   1:  PR[GP1:91,2] = PR[GP1:90,2] + -27.473;
   1:L PR[91] R[100]mm/sec CNT100;
   1:  PR[GP1:91,1] = PR[GP1:90,1] + 0.138;
   1:  PR[GP1:91,2] = PR[GP1:90,2] + -27.866;
   1:L PR[91] R[100]mm/sec CNT100;
   1:  PR[GP1:91,1] = PR[GP1:90,1] + 2.042;
   1:  PR[GP1:91,2] = PR[GP1:90,2] + -27.743;
   1:L PR[91] R[100]mm/sec CNT100;
   1:  PR[GP1:91,1] = PR[GP1:90,1] + 3.999;
   1:  PR[GP1:91,2] = PR[GP1:90,2] + -27.362;
   1:L PR[91] R[100]mm/sec CNT100;
   1:  PR[GP1:91,1] = PR[GP1:90,1] + 7.084;
   1:  PR[GP1:91,2] = PR[GP1:90,2] + -26.955;
   1:L PR[91] R[100]mm/sec CNT100;
   1:  PR[GP1:91,1] = PR[GP1:90,1] + 10.547;
   1:  PR[GP1:91,2] = PR[GP1:90,2] + -25.597;
   1:L PR[91] R[100]mm/sec CNT100;
   1:  PR[GP1:91,1] = PR[GP1:90,1] + 13.465;
   1:  PR[GP1:91,2] = PR[GP1:90,2] + -24.388;
   1:L PR[91] R[100]mm/sec CNT100;
   1:  PR[GP1:91,1] = PR[GP1:90,1] + 16.487;
   1:  PR[GP1:91,2] = PR[GP1:90,2] + -22.246;
   1:L PR[91] R[100]mm/sec CNT100;
   1:  PR[GP1:91,1] = PR[GP1:90,1] + 19.071;
   1:  PR[GP1:91,2] = PR[GP1:90,2] + -20.263;
   1:L PR[91] R[100]mm/sec CNT100;
   1:  PR[GP1:91,1] = PR[GP1:90,1] + 21.139;
   1:  PR[GP1:91,2] = PR[GP1:90,2] + -17.946;
   1:L PR[91] R[100]mm/sec CNT100;
   1:  PR[GP1:91,1] = PR[GP1:90,1] + 23.096;
   1:  PR[GP1:91,2] = PR[GP1:90,2] + -15.395;
   1:L PR[91] R[100]mm/sec CNT100;
   1:  PR[GP1:91,1] = PR[GP1:90,1] + 24.605;
   1:  PR[GP1:91,2] = PR[GP1:90,2] + -12.804;
   1:L PR[91] R[100]mm/sec CNT100;
   1:  PR[GP1:91,1] = PR[GP1:90,1] + 25.817;
   1:  PR[GP1:91,2] = PR[GP1:90,2] + -9.880;
   1:L PR[91] R[100]mm/sec CNT100;
   1:  PR[GP1:91,1] = PR[GP1:90,1] + 26.838;
   1:  PR[GP1:91,2] = PR[GP1:90,2] + -6.844;
   1:L PR[91] R[100]mm/sec CNT100;
   1:  PR[GP1:91,1] = PR[GP1:90,1] + 27.222;
   1:  PR[GP1:91,2] = PR[GP1:90,2] + -3.380;
   1:L PR[91] R[100]mm/sec CNT100;
   1:  PR[GP1:91,1] = PR[GP1:90,1] + 27.629;
   1:  PR[GP1:91,2] = PR[GP1:90,2] + -0.292;
   1:L PR[91] R[100]mm/sec CNT100;
   1:  PR[GP1:91,1] = PR[GP1:90,1] + 27.296;
   1:  PR[GP1:91,2] = PR[GP1:90,2] + 2.903;
   1:L PR[91] R[100]mm/sec CNT100;
   1:  PR[GP1:91,1] = PR[GP1:90,1] + 26.887;
   1:  PR[GP1:91,2] = PR[GP1:90,2] + 6.009;
   1:L PR[91] R[100]mm/sec CNT100;
   1:  PR[GP1:91,1] = PR[GP1:90,1] + 25.954;
   1:  PR[GP1:91,2] = PR[GP1:90,2] + 8.948;
   1:L PR[91] R[100]mm/sec CNT100;
   1:  PR[GP1:91,1] = PR[GP1:90,1] + 24.744;
   1:  PR[GP1:91,2] = PR[GP1:90,2] + 11.869;
   1:L PR[91] R[100]mm/sec CNT100;
   1:  PR[GP1:91,1] = PR[GP1:90,1] + 23.230;
   1:  PR[GP1:91,2] = PR[GP1:90,2] + 14.583;
   1:L PR[91] R[100]mm/sec CNT100;
   1:  PR[GP1:91,1] = PR[GP1:90,1] + 21.280;
   1:  PR[GP1:91,2] = PR[GP1:90,2] + 17.124;
   1:L PR[91] R[100]mm/sec CNT100;
   1:  PR[GP1:91,1] = PR[GP1:90,1] + 19.067;
   1:  PR[GP1:91,2] = PR[GP1:90,2] + 19.643;
   1:L PR[91] R[100]mm/sec CNT100;
   1:  PR[GP1:91,1] = PR[GP1:90,1] + 16.487;
   1:  PR[GP1:91,2] = PR[GP1:90,2] + 21.622;
   1:L PR[91] R[100]mm/sec CNT100;
   1:  PR[GP1:91,1] = PR[GP1:90,1] + 13.451;
   1:  PR[GP1:91,2] = PR[GP1:90,2] + 23.772;
   1:L PR[91] R[100]mm/sec CNT100;
   1:  PR[GP1:91,1] = PR[GP1:90,1] + 10.457;
   1:  PR[GP1:91,2] = PR[GP1:90,2] + 25.012;
   1:L PR[91] R[100]mm/sec CNT100;
   1:  PR[GP1:91,1] = PR[GP1:90,1] + 6.989;
   1:  PR[GP1:91,2] = PR[GP1:90,2] + 26.356;
   1:L PR[91] R[100]mm/sec CNT100;
   1:  PR[GP1:91,1] = PR[GP1:90,1] + 3.774;
   1:  PR[GP1:91,2] = PR[GP1:90,2] + 26.779;
   1:L PR[91] R[100]mm/sec CNT100;
   1:  PR[GP1:91,1] = PR[GP1:90,1] + 0.078;
   1:  PR[GP1:91,2] = PR[GP1:90,2] + 27.237;
   1:L PR[91] R[100]mm/sec CNT100;
   1:  PR[91] = PR[90];
   1:  PR[GP1:91,1] = PR[GP1:90,1] + -2.874;
   1:  PR[GP1:91,2] = PR[GP1:90,2] + 26.871;
   1:  PR[GP1:91,3] = PR[GP1:90,3] + 77.775;
   1:L PR[91] R[100]mm/sec CNT100;
   1:  PR[GP1:91,1] = PR[GP1:90,1] + -6.879;
   1:  PR[GP1:91,2] = PR[GP1:90,2] + 26.344;
   1:L PR[91] R[100]mm/sec CNT100;
   1:  PR[GP1:91,1] = PR[GP1:90,1] + -9.647;
   1:  PR[GP1:91,2] = PR[GP1:90,2] + 25.271;
   1:L PR[91] R[100]mm/sec CNT100;
   1:  PR[GP1:91,1] = PR[GP1:90,1] + -13.376;
   1:  PR[GP1:91,2] = PR[GP1:90,2] + 23.726;
   1:L PR[91] R[100]mm/sec CNT100;
   1:  PR[GP1:91,1] = PR[GP1:90,1] + -15.799;
   1:  PR[GP1:91,2] = PR[GP1:90,2] + 22.010;
   1:L PR[91] R[100]mm/sec CNT100;
   1:  PR[GP1:91,1] = PR[GP1:90,1] + -19.016;
   1:  PR[GP1:91,2] = PR[GP1:90,2] + 19.543;
   1:L PR[91] R[100]mm/sec CNT100;
   1:  PR[GP1:91,1] = PR[GP1:90,1] + -20.663;
   1:  PR[GP1:91,2] = PR[GP1:90,2] + 17.697;
   1:L PR[91] R[100]mm/sec CNT100;
   1:  PR[GP1:91,1] = PR[GP1:90,1] + -23.111;
   1:  PR[GP1:91,2] = PR[GP1:90,2] + 14.505;
   1:L PR[91] R[100]mm/sec CNT100;
   1:  PR[GP1:91,1] = PR[GP1:90,1] + -24.313;
   1:  PR[GP1:91,2] = PR[GP1:90,2] + 12.443;
   1:L PR[91] R[100]mm/sec CNT100;
   1:  PR[GP1:91,1] = PR[GP1:90,1] + -25.837;
   1:  PR[GP1:91,2] = PR[GP1:90,2] + 8.764;
   1:L PR[91] R[100]mm/sec CNT100;
   1:  PR[GP1:91,1] = PR[GP1:90,1] + -26.650;
   1:  PR[GP1:91,2] = PR[GP1:90,2] + 6.347;
   1:L PR[91] R[100]mm/sec CNT100;
   1:  PR[GP1:91,1] = PR[GP1:90,1] + -26.957;
   1:  PR[GP1:91,2] = PR[GP1:90,2] + 3.574;
   1:L PR[91] R[100]mm/sec CNT100;
   1:  PR[GP1:91,1] = PR[GP1:90,1] + -27.472;
   1:  PR[GP1:91,2] = PR[GP1:90,2] + -0.332;
   1:L PR[91] R[100]mm/sec CNT100;
   1:  PR[GP1:91,1] = PR[GP1:90,1] + -27.207;
   1:  PR[GP1:91,2] = PR[GP1:90,2] + -2.875;
   1:L PR[91] R[100]mm/sec CNT100;
   1:  PR[GP1:91,1] = PR[GP1:90,1] + -26.691;
   1:  PR[GP1:91,2] = PR[GP1:90,2] + -6.797;
   1:L PR[91] R[100]mm/sec CNT100;
   1:  PR[GP1:91,1] = PR[GP1:90,1] + -25.949;
   1:  PR[GP1:91,2] = PR[GP1:90,2] + -9.137;
   1:L PR[91] R[100]mm/sec CNT100;
   1:  PR[GP1:91,1] = PR[GP1:90,1] + -24.426;
   1:  PR[GP1:91,2] = PR[GP1:90,2] + -12.814;
   1:L PR[91] R[100]mm/sec CNT100;
   1:  PR[GP1:91,1] = PR[GP1:90,1] + -23.218;
   1:  PR[GP1:91,2] = PR[GP1:90,2] + -14.979;
   1:L PR[91] R[100]mm/sec CNT100;
   1:  PR[GP1:91,1] = PR[GP1:90,1] + -20.776;
   1:  PR[GP1:91,2] = PR[GP1:90,2] + -18.162;
   1:L PR[91] R[100]mm/sec CNT100;
   1:  PR[GP1:91,1] = PR[GP1:90,1] + -19.001;
   1:  PR[GP1:91,2] = PR[GP1:90,2] + -20.182;
   1:L PR[91] R[100]mm/sec CNT100;
   1:  PR[GP1:91,1] = PR[GP1:90,1] + -17.808;
   1:  PR[GP1:91,2] = PR[GP1:90,2] + -21.138;
   1:L PR[91] R[100]mm/sec CNT100;
   1:  PR[GP1:91,1] = PR[GP1:90,1] + -14.562;
   1:  PR[GP1:91,2] = PR[GP1:90,2] + -23.628;
   1:L PR[91] R[100]mm/sec CNT100;
   1:  PR[GP1:91,1] = PR[GP1:90,1] + -13.334;
   1:  PR[GP1:91,2] = PR[GP1:90,2] + -24.378;
   1:L PR[91] R[100]mm/sec CNT100;
   1:  PR[GP1:91,1] = PR[GP1:90,1] + -9.628;
   1:  PR[GP1:91,2] = PR[GP1:90,2] + -25.913;
   1:L PR[91] R[100]mm/sec CNT100;
   1:  PR[GP1:91,1] = PR[GP1:90,1] + -6.838;
   1:  PR[GP1:91,2] = PR[GP1:90,2] + -26.978;
   1:L PR[91] R[100]mm/sec CNT100;
   1:  PR[GP1:91,1] = PR[GP1:90,1] + -3.689;
   1:  PR[GP1:91,2] = PR[GP1:90,2] + -27.362;
   1:L PR[91] R[100]mm/sec CNT100;
   1:  PR[GP1:91,1] = PR[GP1:90,1] + 0.136;
   1:  PR[GP1:91,2] = PR[GP1:90,2] + -27.866;
   1:L PR[91] R[100]mm/sec CNT100;
   1:  PR[GP1:91,1] = PR[GP1:90,1] + 1.630;
   1:  PR[GP1:91,2] = PR[GP1:90,2] + -27.769;
   1:L PR[91] R[100]mm/sec CNT100;
   1:  PR[GP1:91,1] = PR[GP1:90,1] + 3.202;
   1:  PR[GP1:91,2] = PR[GP1:90,2] + -27.463;
   1:L PR[91] R[100]mm/sec CNT100;
   1:  PR[GP1:91,1] = PR[GP1:90,1] + 7.110;
   1:  PR[GP1:91,2] = PR[GP1:90,2] + -26.948;
   1:L PR[91] R[100]mm/sec CNT100;
   1:  PR[GP1:91,1] = PR[GP1:90,1] + 9.876;
   1:  PR[GP1:91,2] = PR[GP1:90,2] + -25.864;
   1:L PR[91] R[100]mm/sec CNT100;
   1:  PR[GP1:91,1] = PR[GP1:90,1] + 13.544;
   1:  PR[GP1:91,2] = PR[GP1:90,2] + -24.344;
   1:L PR[91] R[100]mm/sec CNT100;
   1:  PR[GP1:91,1] = PR[GP1:90,1] + 15.956;
   1:  PR[GP1:91,2] = PR[GP1:90,2] + -22.634;
   1:L PR[91] R[100]mm/sec CNT100;
   1:  PR[GP1:91,1] = PR[GP1:90,1] + 19.173;
   1:  PR[GP1:91,2] = PR[GP1:90,2] + -20.167;
   1:L PR[91] R[100]mm/sec CNT100;
   1:  PR[GP1:91,1] = PR[GP1:90,1] + 20.820;
   1:  PR[GP1:91,2] = PR[GP1:90,2] + -18.321;
   1:L PR[91] R[100]mm/sec CNT100;
   1:  PR[GP1:91,1] = PR[GP1:90,1] + 23.269;
   1:  PR[GP1:91,2] = PR[GP1:90,2] + -15.129;
   1:L PR[91] R[100]mm/sec CNT100;
   1:  PR[GP1:91,1] = PR[GP1:90,1] + 24.470;
   1:  PR[GP1:91,2] = PR[GP1:90,2] + -13.066;
   1:L PR[91] R[100]mm/sec CNT100;
   1:  PR[GP1:91,1] = PR[GP1:90,1] + 25.994;
   1:  PR[GP1:91,2] = PR[GP1:90,2] + -9.387;
   1:L PR[91] R[100]mm/sec CNT100;
   1:  PR[GP1:91,1] = PR[GP1:90,1] + 26.807;
   1:  PR[GP1:91,2] = PR[GP1:90,2] + -6.971;
   1:L PR[91] R[100]mm/sec CNT100;
   1:  PR[GP1:91,1] = PR[GP1:90,1] + 27.114;
   1:  PR[GP1:91,2] = PR[GP1:90,2] + -4.198;
   1:L PR[91] R[100]mm/sec CNT100;
   1:  PR[GP1:91,1] = PR[GP1:90,1] + 27.629;
   1:  PR[GP1:91,2] = PR[GP1:90,2] + -0.292;
   1:L PR[91] R[100]mm/sec CNT100;
   1:  PR[GP1:91,1] = PR[GP1:90,1] + 27.364;
   1:  PR[GP1:91,2] = PR[GP1:90,2] + 2.254;
   1:L PR[91] R[100]mm/sec CNT100;
   1:  PR[GP1:91,1] = PR[GP1:90,1] + 26.847;
   1:  PR[GP1:91,2] = PR[GP1:90,2] + 6.176;
   1:L PR[91] R[100]mm/sec CNT100;
   1:  PR[GP1:91,1] = PR[GP1:90,1] + 26.104;
   1:  PR[GP1:91,2] = PR[GP1:90,2] + 8.517;
   1:L PR[91] R[100]mm/sec CNT100;
   1:  PR[GP1:91,1] = PR[GP1:90,1] + 24.581;
   1:  PR[GP1:91,2] = PR[GP1:90,2] + 12.193;
   1:L PR[91] R[100]mm/sec CNT100;
   1:  PR[GP1:91,1] = PR[GP1:90,1] + 23.375;
   1:  PR[GP1:91,2] = PR[GP1:90,2] + 14.355;
   1:L PR[91] R[100]mm/sec CNT100;
   1:  PR[GP1:91,1] = PR[GP1:90,1] + 20.933;
   1:  PR[GP1:91,2] = PR[GP1:90,2] + 17.538;
   1:L PR[91] R[100]mm/sec CNT100;
   1:  PR[GP1:91,1] = PR[GP1:90,1] + 19.168;
   1:  PR[GP1:91,2] = PR[GP1:90,2] + 19.546;
   1:L PR[91] R[100]mm/sec CNT100;
   1:  PR[GP1:91,1] = PR[GP1:90,1] + 15.957;
   1:  PR[GP1:91,2] = PR[GP1:90,2] + 22.010;
   1:L PR[91] R[100]mm/sec CNT100;
   1:  PR[GP1:91,1] = PR[GP1:90,1] + 13.533;
   1:  PR[GP1:91,2] = PR[GP1:90,2] + 23.726;
   1:L PR[91] R[100]mm/sec CNT100;
   1:  PR[GP1:91,1] = PR[GP1:90,1] + 9.804;
   1:  PR[GP1:91,2] = PR[GP1:90,2] + 25.271;
   1:L PR[91] R[100]mm/sec CNT100;
   1:  PR[GP1:91,1] = PR[GP1:90,1] + 7.035;
   1:  PR[GP1:91,2] = PR[GP1:90,2] + 26.344;
   1:L PR[91] R[100]mm/sec CNT100;
   1:  PR[GP1:91,1] = PR[GP1:90,1] + 3.030;
   1:  PR[GP1:91,2] = PR[GP1:90,2] + 26.871;
   1:L PR[91] R[100]mm/sec CNT100;
   1:  PR[GP1:91,1] = PR[GP1:90,1] + 0.078;
   1:  PR[GP1:91,2] = PR[GP1:90,2] + 27.237;
   1:L PR[91] R[100]mm/sec CNT100;
   1:  PR[91] = PR[90];
   1:  PR[GP1:91,1] = PR[GP1:90,1] + -2.130;
   1:  PR[GP1:91,2] = PR[GP1:90,2] + 26.963;
   1:  PR[GP1:91,3] = PR[GP1:90,3] + 78.385;
   1:L PR[91] R[100]mm/sec CNT100;
   1:  PR[GP1:91,1] = PR[GP1:90,1] + -6.924;
   1:  PR[GP1:91,2] = PR[GP1:90,2] + 26.332;
   1:L PR[91] R[100]mm/sec CNT100;
   1:  PR[GP1:91,1] = PR[GP1:90,1] + -8.993;
   1:  PR[GP1:91,2] = PR[GP1:90,2] + 25.530;
   1:L PR[91] R[100]mm/sec CNT100;
   1:  PR[GP1:91,1] = PR[GP1:90,1] + -13.458;
   1:  PR[GP1:91,2] = PR[GP1:90,2] + 23.681;
   1:L PR[91] R[100]mm/sec CNT100;
   1:  PR[GP1:91,1] = PR[GP1:90,1] + -15.269;
   1:  PR[GP1:91,2] = PR[GP1:90,2] + 22.398;
   1:L PR[91] R[100]mm/sec CNT100;
   1:  PR[GP1:91,1] = PR[GP1:90,1] + -19.117;
   1:  PR[GP1:91,2] = PR[GP1:90,2] + 19.446;
   1:L PR[91] R[100]mm/sec CNT100;
   1:  PR[GP1:91,1] = PR[GP1:90,1] + -20.343;
   1:  PR[GP1:91,2] = PR[GP1:90,2] + 18.072;
   1:L PR[91] R[100]mm/sec CNT100;
   1:  PR[GP1:91,1] = PR[GP1:90,1] + -23.284;
   1:  PR[GP1:91,2] = PR[GP1:90,2] + 14.239;
   1:L PR[91] R[100]mm/sec CNT100;
   1:  PR[GP1:91,1] = PR[GP1:90,1] + -24.178;
   1:  PR[GP1:91,2] = PR[GP1:90,2] + 12.705;
   1:L PR[91] R[100]mm/sec CNT100;
   1:  PR[GP1:91,1] = PR[GP1:90,1] + -26.014;
   1:  PR[GP1:91,2] = PR[GP1:90,2] + 8.271;
   1:L PR[91] R[100]mm/sec CNT100;
   1:  PR[GP1:91,1] = PR[GP1:90,1] + -26.619;
   1:  PR[GP1:91,2] = PR[GP1:90,2] + 6.474;
   1:L PR[91] R[100]mm/sec CNT100;
   1:  PR[GP1:91,1] = PR[GP1:90,1] + -26.849;
   1:  PR[GP1:91,2] = PR[GP1:90,2] + 4.392;
   1:L PR[91] R[100]mm/sec CNT100;
   1:  PR[GP1:91,1] = PR[GP1:90,1] + -27.472;
   1:  PR[GP1:91,2] = PR[GP1:90,2] + -0.332;
   1:L PR[91] R[100]mm/sec CNT100;
   1:  PR[GP1:91,1] = PR[GP1:90,1] + -27.275;
   1:  PR[GP1:91,2] = PR[GP1:90,2] + -2.227;
   1:L PR[91] R[100]mm/sec CNT100;
   1:  PR[GP1:91,1] = PR[GP1:90,1] + -26.651;
   1:  PR[GP1:91,2] = PR[GP1:90,2] + -6.965;
   1:L PR[91] R[100]mm/sec CNT100;
   1:  PR[GP1:91,1] = PR[GP1:90,1] + -26.098;
   1:  PR[GP1:91,2] = PR[GP1:90,2] + -8.707;
   1:L PR[91] R[100]mm/sec CNT100;
   1:  PR[GP1:91,1] = PR[GP1:90,1] + -24.263;
   1:  PR[GP1:91,2] = PR[GP1:90,2] + -13.139;
   1:L PR[91] R[100]mm/sec CNT100;
   1:  PR[GP1:91,1] = PR[GP1:90,1] + -23.363;
   1:  PR[GP1:91,2] = PR[GP1:90,2] + -14.751;
   1:L PR[91] R[100]mm/sec CNT100;
   1:  PR[GP1:91,1] = PR[GP1:90,1] + -20.429;
   1:  PR[GP1:91,2] = PR[GP1:90,2] + -18.575;
   1:L PR[91] R[100]mm/sec CNT100;
   1:  PR[GP1:91,1] = PR[GP1:90,1] + -19.103;
   1:  PR[GP1:91,2] = PR[GP1:90,2] + -20.085;
   1:L PR[91] R[100]mm/sec CNT100;
   1:  PR[GP1:91,1] = PR[GP1:90,1] + -18.219;
   1:  PR[GP1:91,2] = PR[GP1:90,2] + -20.793;
   1:L PR[91] R[100]mm/sec CNT100;
   1:  PR[GP1:91,1] = PR[GP1:90,1] + -14.335;
   1:  PR[GP1:91,2] = PR[GP1:90,2] + -23.773;
   1:L PR[91] R[100]mm/sec CNT100;
   1:  PR[GP1:91,1] = PR[GP1:90,1] + -13.436;
   1:  PR[GP1:91,2] = PR[GP1:90,2] + -24.322;
   1:L PR[91] R[100]mm/sec CNT100;
   1:  PR[GP1:91,1] = PR[GP1:90,1] + -8.980;
   1:  PR[GP1:91,2] = PR[GP1:90,2] + -26.168;
   1:L PR[91] R[100]mm/sec CNT100;
   1:  PR[GP1:91,1] = PR[GP1:90,1] + -6.895;
   1:  PR[GP1:91,2] = PR[GP1:90,2] + -26.963;
   1:L PR[91] R[100]mm/sec CNT100;
   1:  PR[GP1:91,1] = PR[GP1:90,1] + -4.533;
   1:  PR[GP1:91,2] = PR[GP1:90,2] + -27.251;
   1:L PR[91] R[100]mm/sec CNT100;
   1:  PR[GP1:91,1] = PR[GP1:90,1] + 0.134;
   1:  PR[GP1:91,2] = PR[GP1:90,2] + -27.866;
   1:L PR[91] R[100]mm/sec CNT100;
   1:  PR[GP1:91,1] = PR[GP1:90,1] + 1.218;
   1:  PR[GP1:91,2] = PR[GP1:90,2] + -27.796;
   1:L PR[91] R[100]mm/sec CNT100;
   1:  PR[GP1:91,1] = PR[GP1:90,1] + 2.406;
   1:  PR[GP1:91,2] = PR[GP1:90,2] + -27.564;
   1:L PR[91] R[100]mm/sec CNT100;
   1:  PR[GP1:91,1] = PR[GP1:90,1] + 7.137;
   1:  PR[GP1:91,2] = PR[GP1:90,2] + -26.941;
   1:L PR[91] R[100]mm/sec CNT100;
   1:  PR[GP1:91,1] = PR[GP1:90,1] + 9.204;
   1:  PR[GP1:91,2] = PR[GP1:90,2] + -26.131;
   1:L PR[91] R[100]mm/sec CNT100;
   1:  PR[GP1:91,1] = PR[GP1:90,1] + 13.623;
   1:  PR[GP1:91,2] = PR[GP1:90,2] + -24.300;
   1:L PR[91] R[100]mm/sec CNT100;
   1:  PR[GP1:91,1] = PR[GP1:90,1] + 15.426;
   1:  PR[GP1:91,2] = PR[GP1:90,2] + -23.022;
   1:L PR[91] R[100]mm/sec CNT100;
   1:  PR[GP1:91,1] = PR[GP1:90,1] + 19.274;
   1:  PR[GP1:91,2] = PR[GP1:90,2] + -20.070;
   1:L PR[91] R[100]mm/sec CNT100;
   1:  PR[GP1:91,1] = PR[GP1:90,1] + 20.500;
   1:  PR[GP1:91,2] = PR[GP1:90,2] + -18.695;
   1:L PR[91] R[100]mm/sec CNT100;
   1:  PR[GP1:91,1] = PR[GP1:90,1] + 23.441;
   1:  PR[GP1:91,2] = PR[GP1:90,2] + -14.863;
   1:L PR[91] R[100]mm/sec CNT100;
   1:  PR[GP1:91,1] = PR[GP1:90,1] + 24.335;
   1:  PR[GP1:91,2] = PR[GP1:90,2] + -13.328;
   1:L PR[91] R[100]mm/sec CNT100;
   1:  PR[GP1:91,1] = PR[GP1:90,1] + 26.171;
   1:  PR[GP1:91,2] = PR[GP1:90,2] + -8.895;
   1:L PR[91] R[100]mm/sec CNT100;
   1:  PR[GP1:91,1] = PR[GP1:90,1] + 26.776;
   1:  PR[GP1:91,2] = PR[GP1:90,2] + -7.098;
   1:L PR[91] R[100]mm/sec CNT100;
   1:  PR[GP1:91,1] = PR[GP1:90,1] + 27.006;
   1:  PR[GP1:91,2] = PR[GP1:90,2] + -5.016;
   1:L PR[91] R[100]mm/sec CNT100;
   1:  PR[GP1:91,1] = PR[GP1:90,1] + 27.629;
   1:  PR[GP1:91,2] = PR[GP1:90,2] + -0.292;
   1:L PR[91] R[100]mm/sec CNT100;
   1:  PR[GP1:91,1] = PR[GP1:90,1] + 27.431;
   1:  PR[GP1:91,2] = PR[GP1:90,2] + 1.605;
   1:L PR[91] R[100]mm/sec CNT100;
   1:  PR[GP1:91,1] = PR[GP1:90,1] + 26.807;
   1:  PR[GP1:91,2] = PR[GP1:90,2] + 6.343;
   1:L PR[91] R[100]mm/sec CNT100;
   1:  PR[GP1:91,1] = PR[GP1:90,1] + 26.254;
   1:  PR[GP1:91,2] = PR[GP1:90,2] + 8.086;
   1:L PR[91] R[100]mm/sec CNT100;
   1:  PR[GP1:91,1] = PR[GP1:90,1] + 24.418;
   1:  PR[GP1:91,2] = PR[GP1:90,2] + 12.517;
   1:L PR[91] R[100]mm/sec CNT100;
   1:  PR[GP1:91,1] = PR[GP1:90,1] + 23.520;
   1:  PR[GP1:91,2] = PR[GP1:90,2] + 14.126;
   1:L PR[91] R[100]mm/sec CNT100;
   1:  PR[GP1:91,1] = PR[GP1:90,1] + 20.586;
   1:  PR[GP1:91,2] = PR[GP1:90,2] + 17.951;
   1:L PR[91] R[100]mm/sec CNT100;
   1:  PR[GP1:91,1] = PR[GP1:90,1] + 19.270;
   1:  PR[GP1:91,2] = PR[GP1:90,2] + 19.449;
   1:L PR[91] R[100]mm/sec CNT100;
   1:  PR[GP1:91,1] = PR[GP1:90,1] + 15.427;
   1:  PR[GP1:91,2] = PR[GP1:90,2] + 22.398;
   1:L PR[91] R[100]mm/sec CNT100;
   1:  PR[GP1:91,1] = PR[GP1:90,1] + 13.615;
   1:  PR[GP1:91,2] = PR[GP1:90,2] + 23.681;
   1:L PR[91] R[100]mm/sec CNT100;
   1:  PR[GP1:91,1] = PR[GP1:90,1] + 9.150;
   1:  PR[GP1:91,2] = PR[GP1:90,2] + 25.530;
   1:L PR[91] R[100]mm/sec CNT100;
   1:  PR[GP1:91,1] = PR[GP1:90,1] + 7.080;
   1:  PR[GP1:91,2] = PR[GP1:90,2] + 26.332;
   1:L PR[91] R[100]mm/sec CNT100;
   1:  PR[GP1:91,1] = PR[GP1:90,1] + 2.286;
   1:  PR[GP1:91,2] = PR[GP1:90,2] + 26.964;
   1:L PR[91] R[100]mm/sec CNT100;
   1:  PR[GP1:91,1] = PR[GP1:90,1] + 0.078;
   1:  PR[GP1:91,2] = PR[GP1:90,2] + 27.237;
   1:L PR[91] R[100]mm/sec CNT100;
   1:  PR[91] = PR[90];
   1:  PR[GP1:91,1] = PR[GP1:90,1] + -1.386;
   1:  PR[GP1:91,2] = PR[GP1:90,2] + 27.056;
   1:  PR[GP1:91,3] = PR[GP1:90,3] + 78.995;
   1:L PR[91] R[100]mm/sec CNT100;
   1:  PR[GP1:91,1] = PR[GP1:90,1] + -6.969;
   1:  PR[GP1:91,2] = PR[GP1:90,2] + 26.320;
   1:L PR[91] R[100]mm/sec CNT100;
   1:  PR[GP1:91,1] = PR[GP1:90,1] + -8.340;
   1:  PR[GP1:91,2] = PR[GP1:90,2] + 25.789;
   1:L PR[91] R[100]mm/sec CNT100;
   1:  PR[GP1:91,1] = PR[GP1:90,1] + -13.539;
   1:  PR[GP1:91,2] = PR[GP1:90,2] + 23.635;
   1:L PR[91] R[100]mm/sec CNT100;
   1:  PR[GP1:91,1] = PR[GP1:90,1] + -14.739;
   1:  PR[GP1:91,2] = PR[GP1:90,2] + 22.786;
   1:L PR[91] R[100]mm/sec CNT100;
   1:  PR[GP1:91,1] = PR[GP1:90,1] + -19.219;
   1:  PR[GP1:91,2] = PR[GP1:90,2] + 19.349;
   1:L PR[91] R[100]mm/sec CNT100;
   1:  PR[GP1:91,1] = PR[GP1:90,1] + -20.024;
   1:  PR[GP1:91,2] = PR[GP1:90,2] + 18.446;
   1:L PR[91] R[100]mm/sec CNT100;
   1:  PR[GP1:91,1] = PR[GP1:90,1] + -23.457;
   1:  PR[GP1:91,2] = PR[GP1:90,2] + 13.973;
   1:L PR[91] R[100]mm/sec CNT100;
   1:  PR[GP1:91,1] = PR[GP1:90,1] + -24.043;
   1:  PR[GP1:91,2] = PR[GP1:90,2] + 12.966;
   1:L PR[91] R[100]mm/sec CNT100;
   1:  PR[GP1:91,1] = PR[GP1:90,1] + -26.191;
   1:  PR[GP1:91,2] = PR[GP1:90,2] + 7.779;
   1:L PR[91] R[100]mm/sec CNT100;
   1:  PR[GP1:91,1] = PR[GP1:90,1] + -26.588;
   1:  PR[GP1:91,2] = PR[GP1:90,2] + 6.601;
   1:L PR[91] R[100]mm/sec CNT100;
   1:  PR[GP1:91,1] = PR[GP1:90,1] + -26.742;
   1:  PR[GP1:91,2] = PR[GP1:90,2] + 5.211;
   1:L PR[91] R[100]mm/sec CNT100;
   1:  PR[GP1:91,1] = PR[GP1:90,1] + -27.472;
   1:  PR[GP1:91,2] = PR[GP1:90,2] + -0.332;
   1:L PR[91] R[100]mm/sec CNT100;
   1:  PR[GP1:91,1] = PR[GP1:90,1] + -27.342;
   1:  PR[GP1:91,2] = PR[GP1:90,2] + -1.578;
   1:L PR[91] R[100]mm/sec CNT100;
   1:  PR[GP1:91,1] = PR[GP1:90,1] + -26.611;
   1:  PR[GP1:91,2] = PR[GP1:90,2] + -7.133;
   1:L PR[91] R[100]mm/sec CNT100;
   1:  PR[GP1:91,1] = PR[GP1:90,1] + -26.248;
   1:  PR[GP1:91,2] = PR[GP1:90,2] + -8.277;
   1:L PR[91] R[100]mm/sec CNT100;
   1:  PR[GP1:91,1] = PR[GP1:90,1] + -24.100;
   1:  PR[GP1:91,2] = PR[GP1:90,2] + -13.463;
   1:L PR[91] R[100]mm/sec CNT100;
   1:  PR[GP1:91,1] = PR[GP1:90,1] + -23.508;
   1:  PR[GP1:91,2] = PR[GP1:90,2] + -14.523;
   1:L PR[91] R[100]mm/sec CNT100;
   1:  PR[GP1:91,1] = PR[GP1:90,1] + -20.082;
   1:  PR[GP1:91,2] = PR[GP1:90,2] + -18.989;
   1:L PR[91] R[100]mm/sec CNT100;
   1:  PR[GP1:91,1] = PR[GP1:90,1] + -19.204;
   1:  PR[GP1:91,2] = PR[GP1:90,2] + -19.988;
   1:L PR[91] R[100]mm/sec CNT100;
   1:  PR[GP1:91,1] = PR[GP1:90,1] + -18.630;
   1:  PR[GP1:91,2] = PR[GP1:90,2] + -20.448;
   1:L PR[91] R[100]mm/sec CNT100;
   1:  PR[GP1:91,1] = PR[GP1:90,1] + -14.107;
   1:  PR[GP1:91,2] = PR[GP1:90,2] + -23.918;
   1:L PR[91] R[100]mm/sec CNT100;
   1:  PR[GP1:91,1] = PR[GP1:90,1] + -13.539;
   1:  PR[GP1:91,2] = PR[GP1:90,2] + -24.265;
   1:L PR[91] R[100]mm/sec CNT100;
   1:  PR[GP1:91,1] = PR[GP1:90,1] + -8.331;
   1:  PR[GP1:91,2] = PR[GP1:90,2] + -26.422;
   1:L PR[91] R[100]mm/sec CNT100;
   1:  PR[GP1:91,1] = PR[GP1:90,1] + -6.953;
   1:  PR[GP1:91,2] = PR[GP1:90,2] + -26.948;
   1:L PR[91] R[100]mm/sec CNT100;
   1:  PR[GP1:91,1] = PR[GP1:90,1] + -5.378;
   1:  PR[GP1:91,2] = PR[GP1:90,2] + -27.140;
   1:L PR[91] R[100]mm/sec CNT100;
   1:  PR[GP1:91,1] = PR[GP1:90,1] + 0.131;
   1:  PR[GP1:91,2] = PR[GP1:90,2] + -27.866;
   1:L PR[91] R[100]mm/sec CNT100;
   1:  PR[GP1:91,1] = PR[GP1:90,1] + 0.806;
   1:  PR[GP1:91,2] = PR[GP1:90,2] + -27.822;
   1:L PR[91] R[100]mm/sec CNT100;
   1:  PR[GP1:91,1] = PR[GP1:90,1] + 1.609;
   1:  PR[GP1:91,2] = PR[GP1:90,2] + -27.666;
   1:L PR[91] R[100]mm/sec CNT100;
   1:  PR[GP1:91,1] = PR[GP1:90,1] + 7.164;
   1:  PR[GP1:91,2] = PR[GP1:90,2] + -26.934;
   1:L PR[91] R[100]mm/sec CNT100;
   1:  PR[GP1:91,1] = PR[GP1:90,1] + 8.532;
   1:  PR[GP1:91,2] = PR[GP1:90,2] + -26.397;
   1:L PR[91] R[100]mm/sec CNT100;
   1:  PR[GP1:91,1] = PR[GP1:90,1] + 13.702;
   1:  PR[GP1:91,2] = PR[GP1:90,2] + -24.256;
   1:L PR[91] R[100]mm/sec CNT100;
   1:  PR[GP1:91,1] = PR[GP1:90,1] + 14.896;
   1:  PR[GP1:91,2] = PR[GP1:90,2] + -23.410;
   1:L PR[91] R[100]mm/sec CNT100;
   1:  PR[GP1:91,1] = PR[GP1:90,1] + 19.376;
   1:  PR[GP1:91,2] = PR[GP1:90,2] + -19.973;
   1:L PR[91] R[100]mm/sec CNT100;
   1:  PR[GP1:91,1] = PR[GP1:90,1] + 20.181;
   1:  PR[GP1:91,2] = PR[GP1:90,2] + -19.070;
   1:L PR[91] R[100]mm/sec CNT100;
   1:  PR[GP1:91,1] = PR[GP1:90,1] + 23.614;
   1:  PR[GP1:91,2] = PR[GP1:90,2] + -14.596;
   1:L PR[91] R[100]mm/sec CNT100;
   1:  PR[GP1:91,1] = PR[GP1:90,1] + 24.200;
   1:  PR[GP1:91,2] = PR[GP1:90,2] + -13.590;
   1:L PR[91] R[100]mm/sec CNT100;
   1:  PR[GP1:91,1] = PR[GP1:90,1] + 26.348;
   1:  PR[GP1:91,2] = PR[GP1:90,2] + -8.403;
   1:L PR[91] R[100]mm/sec CNT100;
   1:  PR[GP1:91,1] = PR[GP1:90,1] + 26.745;
   1:  PR[GP1:91,2] = PR[GP1:90,2] + -7.225;
   1:L PR[91] R[100]mm/sec CNT100;
   1:  PR[GP1:91,1] = PR[GP1:90,1] + 26.898;
   1:  PR[GP1:91,2] = PR[GP1:90,2] + -5.835;
   1:L PR[91] R[100]mm/sec CNT100;
   1:  PR[GP1:91,1] = PR[GP1:90,1] + 27.629;
   1:  PR[GP1:91,2] = PR[GP1:90,2] + -0.292;
   1:L PR[91] R[100]mm/sec CNT100;
   1:  PR[GP1:91,1] = PR[GP1:90,1] + 27.499;
   1:  PR[GP1:91,2] = PR[GP1:90,2] + 0.956;
   1:L PR[91] R[100]mm/sec CNT100;
   1:  PR[GP1:91,1] = PR[GP1:90,1] + 26.767;
   1:  PR[GP1:91,2] = PR[GP1:90,2] + 6.511;
   1:L PR[91] R[100]mm/sec CNT100;
   1:  PR[GP1:91,1] = PR[GP1:90,1] + 26.404;
   1:  PR[GP1:91,2] = PR[GP1:90,2] + 7.655;
   1:L PR[91] R[100]mm/sec CNT100;
   1:  PR[GP1:91,1] = PR[GP1:90,1] + 24.256;
   1:  PR[GP1:91,2] = PR[GP1:90,2] + 12.841;
   1:L PR[91] R[100]mm/sec CNT100;
   1:  PR[GP1:91,1] = PR[GP1:90,1] + 23.666;
   1:  PR[GP1:91,2] = PR[GP1:90,2] + 13.898;
   1:L PR[91] R[100]mm/sec CNT100;
   1:  PR[GP1:91,1] = PR[GP1:90,1] + 20.239;
   1:  PR[GP1:91,2] = PR[GP1:90,2] + 18.364;
   1:L PR[91] R[100]mm/sec CNT100;
   1:  PR[GP1:91,1] = PR[GP1:90,1] + 19.371;
   1:  PR[GP1:91,2] = PR[GP1:90,2] + 19.352;
   1:L PR[91] R[100]mm/sec CNT100;
   1:  PR[GP1:91,1] = PR[GP1:90,1] + 14.896;
   1:  PR[GP1:91,2] = PR[GP1:90,2] + 22.785;
   1:L PR[91] R[100]mm/sec CNT100;
   1:  PR[GP1:91,1] = PR[GP1:90,1] + 13.696;
   1:  PR[GP1:91,2] = PR[GP1:90,2] + 23.635;
   1:L PR[91] R[100]mm/sec CNT100;
   1:  PR[GP1:91,1] = PR[GP1:90,1] + 8.496;
   1:  PR[GP1:91,2] = PR[GP1:90,2] + 25.789;
   1:L PR[91] R[100]mm/sec CNT100;
   1:  PR[GP1:91,1] = PR[GP1:90,1] + 7.126;
   1:  PR[GP1:91,2] = PR[GP1:90,2] + 26.320;
   1:L PR[91] R[100]mm/sec CNT100;
   1:  PR[GP1:91,1] = PR[GP1:90,1] + 1.542;
   1:  PR[GP1:91,2] = PR[GP1:90,2] + 27.056;
   1:L PR[91] R[100]mm/sec CNT100;
   1:  PR[GP1:91,1] = PR[GP1:90,1] + 0.078;
   1:  PR[GP1:91,2] = PR[GP1:90,2] + 27.237;
   1:L PR[91] R[100]mm/sec CNT100;
   1:  PR[91] = PR[90];
   1:  PR[GP1:91,1] = PR[GP1:90,1] + -0.641;
   1:  PR[GP1:91,2] = PR[GP1:90,2] + 27.148;
   1:  PR[GP1:91,3] = PR[GP1:90,3] + 79.605;
   1:L PR[91] R[100]mm/sec CNT100;
   1:  PR[GP1:91,1] = PR[GP1:90,1] + -7.014;
   1:  PR[GP1:91,2] = PR[GP1:90,2] + 26.308;
   1:L PR[91] R[100]mm/sec CNT100;
   1:  PR[GP1:91,1] = PR[GP1:90,1] + -7.686;
   1:  PR[GP1:91,2] = PR[GP1:90,2] + 26.048;
   1:L PR[91] R[100]mm/sec CNT100;
   1:  PR[GP1:91,1] = PR[GP1:90,1] + -13.621;
   1:  PR[GP1:91,2] = PR[GP1:90,2] + 23.590;
   1:L PR[91] R[100]mm/sec CNT100;
   1:  PR[GP1:91,1] = PR[GP1:90,1] + -14.209;
   1:  PR[GP1:91,2] = PR[GP1:90,2] + 23.173;
   1:L PR[91] R[100]mm/sec CNT100;
   1:  PR[GP1:91,1] = PR[GP1:90,1] + -19.320;
   1:  PR[GP1:91,2] = PR[GP1:90,2] + 19.252;
   1:L PR[91] R[100]mm/sec CNT100;
   1:  PR[GP1:91,1] = PR[GP1:90,1] + -19.705;
   1:  PR[GP1:91,2] = PR[GP1:90,2] + 18.821;
   1:L PR[91] R[100]mm/sec CNT100;
   1:  PR[GP1:91,1] = PR[GP1:90,1] + -23.629;
   1:  PR[GP1:91,2] = PR[GP1:90,2] + 13.706;
   1:L PR[91] R[100]mm/sec CNT100;
   1:  PR[GP1:91,1] = PR[GP1:90,1] + -23.908;
   1:  PR[GP1:91,2] = PR[GP1:90,2] + 13.228;
   1:L PR[91] R[100]mm/sec CNT100;
   1:  PR[GP1:91,1] = PR[GP1:90,1] + -26.369;
   1:  PR[GP1:91,2] = PR[GP1:90,2] + 7.287;
   1:L PR[91] R[100]mm/sec CNT100;
   1:  PR[GP1:91,1] = PR[GP1:90,1] + -26.556;
   1:  PR[GP1:91,2] = PR[GP1:90,2] + 6.728;
   1:L PR[91] R[100]mm/sec CNT100;
   1:  PR[GP1:91,1] = PR[GP1:90,1] + -26.634;
   1:  PR[GP1:91,2] = PR[GP1:90,2] + 6.029;
   1:L PR[91] R[100]mm/sec CNT100;
   1:  PR[GP1:91,1] = PR[GP1:90,1] + -27.472;
   1:  PR[GP1:91,2] = PR[GP1:90,2] + -0.332;
   1:L PR[91] R[100]mm/sec CNT100;
   1:  PR[GP1:91,1] = PR[GP1:90,1] + -27.410;
   1:  PR[GP1:91,2] = PR[GP1:90,2] + -0.930;
   1:L PR[91] R[100]mm/sec CNT100;
   1:  PR[GP1:91,1] = PR[GP1:90,1] + -26.570;
   1:  PR[GP1:91,2] = PR[GP1:90,2] + -7.301;
   1:L PR[91] R[100]mm/sec CNT100;
   1:  PR[GP1:91,1] = PR[GP1:90,1] + -26.397;
   1:  PR[GP1:91,2] = PR[GP1:90,2] + -7.847;
   1:L PR[91] R[100]mm/sec CNT100;
   1:  PR[GP1:91,1] = PR[GP1:90,1] + -23.936;
   1:  PR[GP1:91,2] = PR[GP1:90,2] + -13.788;
   1:L PR[91] R[100]mm/sec CNT100;
   1:  PR[GP1:91,1] = PR[GP1:90,1] + -23.654;
   1:  PR[GP1:91,2] = PR[GP1:90,2] + -14.294;
   1:L PR[91] R[100]mm/sec CNT100;
   1:  PR[GP1:91,1] = PR[GP1:90,1] + -19.735;
   1:  PR[GP1:91,2] = PR[GP1:90,2] + -19.402;
   1:L PR[91] R[100]mm/sec CNT100;
   1:  PR[GP1:91,1] = PR[GP1:90,1] + -19.306;
   1:  PR[GP1:91,2] = PR[GP1:90,2] + -19.891;
   1:L PR[91] R[100]mm/sec CNT100;
   1:  PR[GP1:91,1] = PR[GP1:90,1] + -19.040;
   1:  PR[GP1:91,2] = PR[GP1:90,2] + -20.103;
   1:L PR[91] R[100]mm/sec CNT100;
   1:  PR[GP1:91,1] = PR[GP1:90,1] + -13.880;
   1:  PR[GP1:91,2] = PR[GP1:90,2] + -24.062;
   1:L PR[91] R[100]mm/sec CNT100;
   1:  PR[GP1:91,1] = PR[GP1:90,1] + -13.641;
   1:  PR[GP1:91,2] = PR[GP1:90,2] + -24.208;
   1:L PR[91] R[100]mm/sec CNT100;
   1:  PR[GP1:91,1] = PR[GP1:90,1] + -7.683;
   1:  PR[GP1:91,2] = PR[GP1:90,2] + -26.676;
   1:L PR[91] R[100]mm/sec CNT100;
   1:  PR[GP1:91,1] = PR[GP1:90,1] + -7.004;
   1:  PR[GP1:91,2] = PR[GP1:90,2] + -26.935;
   1:L PR[91] R[100]mm/sec CNT100;
   1:  PR[GP1:91,1] = PR[GP1:90,1] + 0.128;
   1:  PR[GP1:91,2] = PR[GP1:90,2] + -27.866;
   1:L PR[91] R[100]mm/sec CNT100;
   1:  PR[GP1:91,1] = PR[GP1:90,1] + 0.394;
   1:  PR[GP1:91,2] = PR[GP1:90,2] + -27.849;
   1:L PR[91] R[100]mm/sec CNT100;
   1:  PR[GP1:91,1] = PR[GP1:90,1] + 0.813;
   1:  PR[GP1:91,2] = PR[GP1:90,2] + -27.767;
   1:L PR[91] R[100]mm/sec CNT100;
   1:  PR[GP1:91,1] = PR[GP1:90,1] + 7.191;
   1:  PR[GP1:91,2] = PR[GP1:90,2] + -26.927;
   1:L PR[91] R[100]mm/sec CNT100;
   1:  PR[GP1:91,1] = PR[GP1:90,1] + 7.862;
   1:  PR[GP1:91,2] = PR[GP1:90,2] + -26.664;
   1:L PR[91] R[100]mm/sec CNT100;
   1:  PR[GP1:91,1] = PR[GP1:90,1] + 13.781;
   1:  PR[GP1:91,2] = PR[GP1:90,2] + -24.212;
   1:L PR[91] R[100]mm/sec CNT100;
   1:  PR[GP1:91,1] = PR[GP1:90,1] + 14.365;
   1:  PR[GP1:91,2] = PR[GP1:90,2] + -23.798;
   1:L PR[91] R[100]mm/sec CNT100;
   1:  PR[GP1:91,1] = PR[GP1:90,1] + 19.477;
   1:  PR[GP1:91,2] = PR[GP1:90,2] + -19.876;
   1:L PR[91] R[100]mm/sec CNT100;
   1:  PR[GP1:91,1] = PR[GP1:90,1] + 19.862;
   1:  PR[GP1:91,2] = PR[GP1:90,2] + -19.445;
   1:L PR[91] R[100]mm/sec CNT100;
   1:  PR[GP1:91,1] = PR[GP1:90,1] + 23.786;
   1:  PR[GP1:91,2] = PR[GP1:90,2] + -14.330;
   1:L PR[91] R[100]mm/sec CNT100;
   1:  PR[GP1:91,1] = PR[GP1:90,1] + 24.064;
   1:  PR[GP1:91,2] = PR[GP1:90,2] + -13.852;
   1:L PR[91] R[100]mm/sec CNT100;
   1:  PR[GP1:91,1] = PR[GP1:90,1] + 26.525;
   1:  PR[GP1:91,2] = PR[GP1:90,2] + -7.910;
   1:L PR[91] R[100]mm/sec CNT100;
   1:  PR[GP1:91,1] = PR[GP1:90,1] + 26.713;
   1:  PR[GP1:91,2] = PR[GP1:90,2] + -7.352;
   1:L PR[91] R[100]mm/sec CNT100;
   1:  PR[GP1:91,1] = PR[GP1:90,1] + 26.791;
   1:  PR[GP1:91,2] = PR[GP1:90,2] + -6.653;
   1:L PR[91] R[100]mm/sec CNT100;
   1:  PR[GP1:91,1] = PR[GP1:90,1] + 27.629;
   1:  PR[GP1:91,2] = PR[GP1:90,2] + -0.292;
   1:L PR[91] R[100]mm/sec CNT100;
   1:  PR[GP1:91,1] = PR[GP1:90,1] + 27.566;
   1:  PR[GP1:91,2] = PR[GP1:90,2] + 0.307;
   1:L PR[91] R[100]mm/sec CNT100;
   1:  PR[GP1:91,1] = PR[GP1:90,1] + 26.727;
   1:  PR[GP1:91,2] = PR[GP1:90,2] + 6.678;
   1:L PR[91] R[100]mm/sec CNT100;
   1:  PR[GP1:91,1] = PR[GP1:90,1] + 26.554;
   1:  PR[GP1:91,2] = PR[GP1:90,2] + 7.224;
   1:L PR[91] R[100]mm/sec CNT100;
   1:  PR[GP1:91,1] = PR[GP1:90,1] + 24.093;
   1:  PR[GP1:91,2] = PR[GP1:90,2] + 13.165;
   1:L PR[91] R[100]mm/sec CNT100;
   1:  PR[GP1:91,1] = PR[GP1:90,1] + 23.811;
   1:  PR[GP1:91,2] = PR[GP1:90,2] + 13.670;
   1:L PR[91] R[100]mm/sec CNT100;
   1:  PR[GP1:91,1] = PR[GP1:90,1] + 19.892;
   1:  PR[GP1:91,2] = PR[GP1:90,2] + 18.778;
   1:L PR[91] R[100]mm/sec CNT100;
   1:  PR[GP1:91,1] = PR[GP1:90,1] + 19.473;
   1:  PR[GP1:91,2] = PR[GP1:90,2] + 19.255;
   1:L PR[91] R[100]mm/sec CNT100;
   1:  PR[GP1:91,1] = PR[GP1:90,1] + 14.366;
   1:  PR[GP1:91,2] = PR[GP1:90,2] + 23.173;
   1:L PR[91] R[100]mm/sec CNT100;
   1:  PR[GP1:91,1] = PR[GP1:90,1] + 13.778;
   1:  PR[GP1:91,2] = PR[GP1:90,2] + 23.590;
   1:L PR[91] R[100]mm/sec CNT100;
   1:  PR[GP1:91,1] = PR[GP1:90,1] + 7.843;
   1:  PR[GP1:91,2] = PR[GP1:90,2] + 26.048;
   1:L PR[91] R[100]mm/sec CNT100;
   1:  PR[GP1:91,1] = PR[GP1:90,1] + 7.172;
   1:  PR[GP1:91,2] = PR[GP1:90,2] + 26.308;
   1:L PR[91] R[100]mm/sec CNT100;
   1:  PR[GP1:91,1] = PR[GP1:90,1] + 0.073;
   1:  PR[GP1:91,2] = PR[GP1:90,2] + 27.236;
   1:L PR[91] R[100]mm/sec CNT100;
   1:  PR[91] = PR[90];
   1:  PR[GP1:91,1] = PR[GP1:90,1] + -7.043;
   1:  PR[GP1:91,2] = PR[GP1:90,2] + 26.299;
   1:  PR[GP1:91,3] = PR[GP1:90,3] + 80.215;
   1:L PR[91] R[100]mm/sec CNT100;
   1:  PR[GP1:91,1] = PR[GP1:90,1] + -13.678;
   1:  PR[GP1:91,2] = PR[GP1:90,2] + 23.555;
   1:L PR[91] R[100]mm/sec CNT100;
   1:  PR[GP1:91,1] = PR[GP1:90,1] + -19.380;
   1:  PR[GP1:91,2] = PR[GP1:90,2] + 19.187;
   1:L PR[91] R[100]mm/sec CNT100;
   1:  PR[GP1:91,1] = PR[GP1:90,1] + -23.783;
   1:  PR[GP1:91,2] = PR[GP1:90,2] + 13.463;
   1:L PR[91] R[100]mm/sec CNT100;
   1:  PR[GP1:91,1] = PR[GP1:90,1] + -26.536;
   1:  PR[GP1:91,2] = PR[GP1:90,2] + 6.793;
   1:L PR[91] R[100]mm/sec CNT100;
   1:  PR[GP1:91,1] = PR[GP1:90,1] + -27.469;
   1:  PR[GP1:91,2] = PR[GP1:90,2] + -0.312;
   1:L PR[91] R[100]mm/sec CNT100;
   1:  PR[GP1:91,1] = PR[GP1:90,1] + -26.533;
   1:  PR[GP1:91,2] = PR[GP1:90,2] + -7.451;
   1:L PR[91] R[100]mm/sec CNT100;
   1:  PR[GP1:91,1] = PR[GP1:90,1] + -23.785;
   1:  PR[GP1:91,2] = PR[GP1:90,2] + -14.085;
   1:L PR[91] R[100]mm/sec CNT100;
   1:  PR[GP1:91,1] = PR[GP1:90,1] + -19.416;
   1:  PR[GP1:91,2] = PR[GP1:90,2] + -19.779;
   1:L PR[91] R[100]mm/sec CNT100;
   1:  PR[GP1:91,1] = PR[GP1:90,1] + -19.389;
   1:  PR[GP1:91,2] = PR[GP1:90,2] + -19.806;
   1:L PR[91] R[100]mm/sec CNT100;
   1:  PR[GP1:91,1] = PR[GP1:90,1] + -13.673;
   1:  PR[GP1:91,2] = PR[GP1:90,2] + -24.181;
   1:L PR[91] R[100]mm/sec CNT100;
   1:  PR[GP1:91,1] = PR[GP1:90,1] + -7.041;
   1:  PR[GP1:91,2] = PR[GP1:90,2] + -26.923;
   1:L PR[91] R[100]mm/sec CNT100;
   1:  PR[GP1:91,1] = PR[GP1:90,1] + 0.101;
   1:  PR[GP1:91,2] = PR[GP1:90,2] + -27.862;
   1:L PR[91] R[100]mm/sec CNT100;
   1:  PR[GP1:91,1] = PR[GP1:90,1] + 7.204;
   1:  PR[GP1:91,2] = PR[GP1:90,2] + -26.922;
   1:L PR[91] R[100]mm/sec CNT100;
   1:  PR[GP1:91,1] = PR[GP1:90,1] + 13.835;
   1:  PR[GP1:91,2] = PR[GP1:90,2] + -24.178;
   1:L PR[91] R[100]mm/sec CNT100;
   1:  PR[GP1:91,1] = PR[GP1:90,1] + 19.567;
   1:  PR[GP1:91,2] = PR[GP1:90,2] + -19.788;
   1:L PR[91] R[100]mm/sec CNT100;
   1:  PR[GP1:91,1] = PR[GP1:90,1] + 23.940;
   1:  PR[GP1:91,2] = PR[GP1:90,2] + -14.088;
   1:L PR[91] R[100]mm/sec CNT100;
   1:  PR[GP1:91,1] = PR[GP1:90,1] + 26.688;
   1:  PR[GP1:91,2] = PR[GP1:90,2] + -7.452;
   1:L PR[91] R[100]mm/sec CNT100;
   1:  PR[GP1:91,1] = PR[GP1:90,1] + 27.626;
   1:  PR[GP1:91,2] = PR[GP1:90,2] + -0.312;
   1:L PR[91] R[100]mm/sec CNT100;
   1:  PR[GP1:91,1] = PR[GP1:90,1] + 26.689;
   1:  PR[GP1:91,2] = PR[GP1:90,2] + 6.827;
   1:L PR[91] R[100]mm/sec CNT100;
   1:  PR[GP1:91,1] = PR[GP1:90,1] + 23.942;
   1:  PR[GP1:91,2] = PR[GP1:90,2] + 13.461;
   1:L PR[91] R[100]mm/sec CNT100;
   1:  PR[GP1:91,1] = PR[GP1:90,1] + 19.566;
   1:  PR[GP1:91,2] = PR[GP1:90,2] + 19.165;
   1:L PR[91] R[100]mm/sec CNT100;
   1:  PR[GP1:91,1] = PR[GP1:90,1] + 13.834;
   1:  PR[GP1:91,2] = PR[GP1:90,2] + 23.555;
   1:L PR[91] R[100]mm/sec CNT100;
   1:  PR[GP1:91,1] = PR[GP1:90,1] + 7.200;
   1:  PR[GP1:91,2] = PR[GP1:90,2] + 26.299;
   1:L PR[91] R[100]mm/sec CNT100;
   1:  PR[GP1:91,1] = PR[GP1:90,1] + 0.078;
   1:  PR[GP1:91,2] = PR[GP1:90,2] + 27.237;
   1:L PR[91] R[100]mm/sec CNT100;
   1:  PR[GP1:91,1] = PR[GP1:90,1] + -7.043;
   1:  PR[GP1:91,2] = PR[GP1:90,2] + 26.299;
   1:L PR[91] R[100]mm/sec CNT100;
   1:  PR[GP1:91,1] = PR[GP1:90,1] + -13.678;
   1:  PR[GP1:91,2] = PR[GP1:90,2] + 23.555;
   1:L PR[91] R[100]mm/sec CNT100;
   1:  PR[GP1:91,1] = PR[GP1:90,1] + -19.380;
   1:  PR[GP1:91,2] = PR[GP1:90,2] + 19.187;
   1:L PR[91] R[100]mm/sec CNT100;
   1:  PR[GP1:91,1] = PR[GP1:90,1] + -23.783;
   1:  PR[GP1:91,2] = PR[GP1:90,2] + 13.463;
   1:L PR[91] R[100]mm/sec CNT100;
   1:  PR[GP1:91,1] = PR[GP1:90,1] + -26.536;
   1:  PR[GP1:91,2] = PR[GP1:90,2] + 6.793;
   1:L PR[91] R[100]mm/sec CNT100;
   1:  PR[GP1:91,1] = PR[GP1:90,1] + -27.469;
   1:  PR[GP1:91,2] = PR[GP1:90,2] + -0.312;
   1:L PR[91] R[100]mm/sec CNT100;
   1:  PR[GP1:91,1] = PR[GP1:90,1] + -26.533;
   1:  PR[GP1:91,2] = PR[GP1:90,2] + -7.451;
   1:L PR[91] R[100]mm/sec CNT100;
   1:  PR[GP1:91,1] = PR[GP1:90,1] + -23.785;
   1:  PR[GP1:91,2] = PR[GP1:90,2] + -14.085;
   1:L PR[91] R[100]mm/sec CNT100;
   1:  PR[GP1:91,1] = PR[GP1:90,1] + -19.416;
   1:  PR[GP1:91,2] = PR[GP1:90,2] + -19.779;
   1:L PR[91] R[100]mm/sec CNT100;
   1:  PR[GP1:91,1] = PR[GP1:90,1] + -19.389;
   1:  PR[GP1:91,2] = PR[GP1:90,2] + -19.806;
   1:L PR[91] R[100]mm/sec CNT100;
   1:  PR[GP1:91,1] = PR[GP1:90,1] + -13.673;
   1:  PR[GP1:91,2] = PR[GP1:90,2] + -24.181;
   1:L PR[91] R[100]mm/sec CNT100;
   1:  PR[GP1:91,1] = PR[GP1:90,1] + -7.041;
   1:  PR[GP1:91,2] = PR[GP1:90,2] + -26.923;
   1:L PR[91] R[100]mm/sec CNT100;
   1:  PR[GP1:91,1] = PR[GP1:90,1] + 0.101;
   1:  PR[GP1:91,2] = PR[GP1:90,2] + -27.862;
   1:L PR[91] R[100]mm/sec CNT100;
   1:  PR[GP1:91,1] = PR[GP1:90,1] + 7.204;
   1:  PR[GP1:91,2] = PR[GP1:90,2] + -26.922;
   1:L PR[91] R[100]mm/sec CNT100;
   1:  PR[GP1:91,1] = PR[GP1:90,1] + 13.835;
   1:  PR[GP1:91,2] = PR[GP1:90,2] + -24.178;
   1:L PR[91] R[100]mm/sec CNT100;
   1:  PR[GP1:91,1] = PR[GP1:90,1] + 19.567;
   1:  PR[GP1:91,2] = PR[GP1:90,2] + -19.788;
   1:L PR[91] R[100]mm/sec CNT100;
   1:  PR[GP1:91,1] = PR[GP1:90,1] + 23.940;
   1:  PR[GP1:91,2] = PR[GP1:90,2] + -14.088;
   1:L PR[91] R[100]mm/sec CNT100;
   1:  PR[GP1:91,1] = PR[GP1:90,1] + 26.688;
   1:  PR[GP1:91,2] = PR[GP1:90,2] + -7.452;
   1:L PR[91] R[100]mm/sec CNT100;
   1:  PR[GP1:91,1] = PR[GP1:90,1] + 27.626;
   1:  PR[GP1:91,2] = PR[GP1:90,2] + -0.312;
   1:L PR[91] R[100]mm/sec CNT100;
   1:  PR[GP1:91,1] = PR[GP1:90,1] + 26.689;
   1:  PR[GP1:91,2] = PR[GP1:90,2] + 6.827;
   1:L PR[91] R[100]mm/sec CNT100;
   1:  PR[GP1:91,1] = PR[GP1:90,1] + 23.942;
   1:  PR[GP1:91,2] = PR[GP1:90,2] + 13.461;
   1:L PR[91] R[100]mm/sec CNT100;
   1:  PR[GP1:91,1] = PR[GP1:90,1] + 19.566;
   1:  PR[GP1:91,2] = PR[GP1:90,2] + 19.165;
   1:L PR[91] R[100]mm/sec CNT100;
   1:  PR[GP1:91,1] = PR[GP1:90,1] + 13.834;
   1:  PR[GP1:91,2] = PR[GP1:90,2] + 23.555;
   1:L PR[91] R[100]mm/sec CNT100;
   1:  PR[GP1:91,1] = PR[GP1:90,1] + 7.200;
   1:  PR[GP1:91,2] = PR[GP1:90,2] + 26.299;
   1:L PR[91] R[100]mm/sec CNT100;
   1:  PR[GP1:91,1] = PR[GP1:90,1] + 0.078;
   1:  PR[GP1:91,2] = PR[GP1:90,2] + 27.237;
   1:L PR[91] R[100]mm/sec CNT100 TB   .50sec,CALL END_PUD;
   1:  DO[117:Laser Start]=OFF;
   1:  PR[92] = PR[91];
   1:  PR[GP1:92,3] = PR[GP1:92,3] + 50;
   1:J PR[92] 10% FINE;
   1:  WAIT   5.00(sec);
   1:  DO[119:Gas]=OFF;
   1:  CALL HOME_ALL;
/POS
/END
